(*
SPDX-FileCopyrightText: © 2026 Oleksandr Tiutyk <trofimich@gmail.com>
SPDX-License-Identifier: MIT
License: https://opensource.org/license/mit
*)

INTERFACE IDataMemberNotSpecifiedException EXTENDS IGeneralException

METHOD Throw
VAR_INPUT
	sourceNamespaceName : STRING;
	sourceClassName : STRING;
	sourcePOUName : STRING;
	sourcePosition : STRING;
	dataMemberName : STRING;
END_VAR
END_METHOD

END_INTERFACE

(* stored: Version 1.1.0.1
   Itf IDataMemberNotSpecifiedException: Id {2350b160-aedd-4da5-961b-4f214e2e1cd3}
   Method Throw: Id {f32c598e-d35c-4a9c-a210-c8741838f001} *)
